// TIA Portal V16 export
// export: Created 2024-06-24T15:42:27.9585009Z, ExportSetting WithDefaults, DisplayName Totally Integrated Automation Portal, DisplayVersion V16, DisplayName TIA Portal Version Control Interface, DisplayVersion V16, DisplayName TIA Portal Openness, DisplayVersion V16, DisplayName STEP 7 Professional, DisplayVersion V16, DisplayName STEP 7 Safety, DisplayVersion V16, DisplayName WinCC Advanced, DisplayVersion V16
ORGANIZATION_BLOCK "OB_Master"   // OB124, LAD, ProgramCycle
TITLE = "Main Program Sweep (Cycle)"
{ S7_Optimized_Access := 'TRUE' }
VERSION : 0.1
// stored: AutoNumber true, IsIECCheckEnabled false, SetENOAutomatically false
   VAR_INPUT
      Initial_Call : Bool;   // Initial call of this OB
      Remanence : Bool;   // =True, if remanent data are available
   END_VAR
BEGIN

REGION Network 1
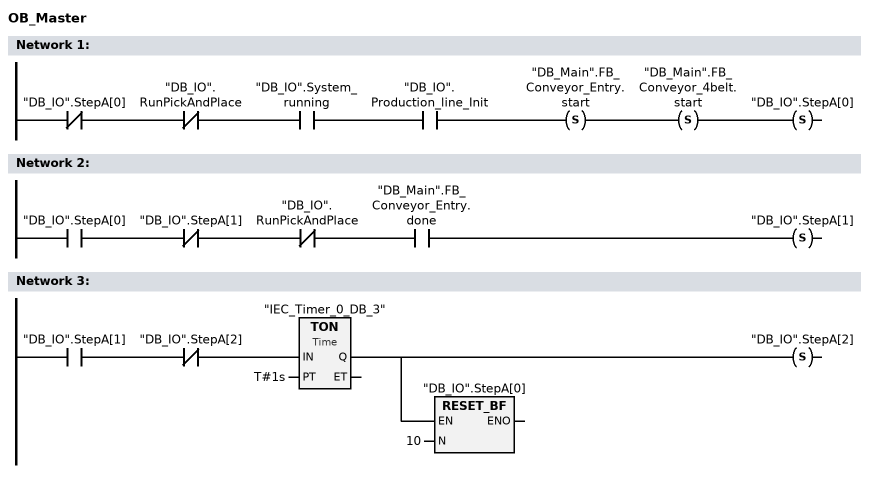
   RUNG wire#powerrail
      I_Contact( "DB_IO".StepA[0] )
      I_Contact( "DB_IO".RunPickAndPlace )
      Contact( "DB_IO".System_running )
      Contact( "DB_IO".Production_line_Init )
      S_Coil( "DB_Main".FB_Conveyor_Entry.start )
      S_Coil( "DB_Main".FB_Conveyor_4belt.start )
      S_Coil( "DB_IO".StepA[0] )
   END_RUNG
   // the same network as SCL:
   IF NOT "DB_IO".StepA[0] AND NOT "DB_IO".RunPickAndPlace AND "DB_IO".System_running AND "DB_IO".Production_line_Init THEN
       "DB_Main".FB_Conveyor_Entry.start := TRUE;
       "DB_Main".FB_Conveyor_4belt.start := TRUE;
       "DB_IO".StepA[0] := TRUE;
   END_IF;
END_REGION

REGION Network 2
   RUNG wire#powerrail
      Contact( "DB_IO".StepA[0] )
      I_Contact( "DB_IO".StepA[1] )
      I_Contact( "DB_IO".RunPickAndPlace )
      Contact( "DB_Main".FB_Conveyor_Entry.done )
      S_Coil( "DB_IO".StepA[1] )
   END_RUNG
   // the same network as SCL:
   IF "DB_IO".StepA[0] AND NOT "DB_IO".StepA[1] AND NOT "DB_IO".RunPickAndPlace AND "DB_Main".FB_Conveyor_Entry.done THEN
       "DB_IO".StepA[1] := TRUE;
   END_IF;
END_REGION

REGION Network 3
   // no SCL statement known for RBitfield: written as a call
   "IEC_Timer_0_DB_3".TON(IN := "DB_IO".StepA[1] AND NOT "DB_IO".StepA[2], PT := T#1s);
   IF "IEC_Timer_0_DB_3".Q THEN
       "DB_IO".StepA[2] := TRUE;
       RESET_BF(operand := "DB_IO".StepA[0], n := 10);
   END_IF;
END_REGION
END_ORGANIZATION_BLOCK
